TYPE STATE:
    STRUCT
        curTime: LREAL;
        dvar_M_p_vt AT %Q*: BOOL;
        dvar_M_p_vf AT %Q*: BOOL;
        dvar_M_p_vr2 AT %Q*: DINT;
        dvar_M_p_vr3 AT %Q*: DINT;
        dvar_M_p_v0 AT %Q*: DINT;
        dvar_M_p_v1 AT %Q*: DINT;
        dvar_M_p_v2 AT %Q*: DINT;
        dvar_M_p_v3 AT %Q*: DINT;
        dvar_M_p_v123 AT %Q*: DINT;
        dvar_M_p_vn1 AT %Q*: DINT;
        dvar_M_p_vn2 AT %Q*: DINT;
        dvar_M_p_v00 AT %Q*: LREAL;
        dvar_M_p_v01 AT %Q*: LREAL;
        dvar_M_p_v05 AT %Q*: LREAL;
        dvar_M_p_v10 AT %Q*: LREAL;
        dvar_M_p_v20 AT %Q*: LREAL;
        dvar_M_p_v30 AT %Q*: LREAL;
        dvar_M_p_v270 AT %Q*: LREAL;
        dvar_M_p_vn01 AT %Q*: LREAL;
        dvar_M_p_vn10 AT %Q*: LREAL;
        dvar_M_p_e AT %Q*: LREAL;
        dvar_M_p_ve1 AT %Q*: enum_E;
        dvar_M_p_ve2 AT %Q*: enum_E;
        dvar_M_p_ve3 AT %Q*: enum_E;
        dvar_M_p_ve4 AT %Q*: enum_E;
        dvar_M_p_vbir AT %Q*: TupleStruct_2;
        dvar_M_p_vb000 AT %Q*: BOOL;
        dvar_M_p_vb001 AT %Q*: BOOL;
        dvar_M_p_vb002 AT %Q*: BOOL;
        dvar_M_p_vb003 AT %Q*: BOOL;
        dvar_M_p_vb004 AT %Q*: BOOL;
        dvar_M_p_vb005 AT %Q*: BOOL;
        dvar_M_p_vb006 AT %Q*: BOOL;
        dvar_M_p_vb007 AT %Q*: BOOL;
        dvar_M_p_vb008 AT %Q*: BOOL;
        dvar_M_p_vb009 AT %Q*: BOOL;
        dvar_M_p_vb010 AT %Q*: BOOL;
        dvar_M_p_vb011 AT %Q*: BOOL;
        dvar_M_p_vb012 AT %Q*: BOOL;
        dvar_M_p_vb013 AT %Q*: BOOL;
        dvar_M_p_vb014 AT %Q*: BOOL;
        dvar_M_p_vb015 AT %Q*: BOOL;
        dvar_M_p_vb016 AT %Q*: BOOL;
        dvar_M_p_vb017 AT %Q*: BOOL;
        dvar_M_p_vb018 AT %Q*: BOOL;
        dvar_M_p_vb019 AT %Q*: BOOL;
        dvar_M_p_vb020 AT %Q*: BOOL;
        dvar_M_p_vb021 AT %Q*: BOOL;
        dvar_M_p_vb022 AT %Q*: BOOL;
        dvar_M_p_vb023 AT %Q*: BOOL;
        dvar_M_p_vb024 AT %Q*: BOOL;
        dvar_M_p_vb025 AT %Q*: BOOL;
        dvar_M_p_vb026 AT %Q*: BOOL;
        dvar_M_p_vb027 AT %Q*: BOOL;
        dvar_M_p_vb028 AT %Q*: BOOL;
        dvar_M_p_vb029 AT %Q*: BOOL;
        dvar_M_p_vb030 AT %Q*: BOOL;
        dvar_M_p_vb031 AT %Q*: BOOL;
        dvar_M_p_vb032 AT %Q*: BOOL;
        dvar_M_p_vb033 AT %Q*: BOOL;
        dvar_M_p_vb034 AT %Q*: BOOL;
        dvar_M_p_vb035 AT %Q*: BOOL;
        dvar_M_p_vb036 AT %Q*: BOOL;
        dvar_M_p_vb037 AT %Q*: BOOL;
        dvar_M_p_vb038 AT %Q*: BOOL;
        dvar_M_p_vb039 AT %Q*: BOOL;
        dvar_M_p_vb040 AT %Q*: BOOL;
        dvar_M_p_vb041 AT %Q*: BOOL;
        dvar_M_p_vb042 AT %Q*: BOOL;
        dvar_M_p_vb043 AT %Q*: BOOL;
        dvar_M_p_vb044 AT %Q*: BOOL;
        dvar_M_p_vb045 AT %Q*: BOOL;
        dvar_M_p_vb046 AT %Q*: BOOL;
        dvar_M_p_vb047 AT %Q*: BOOL;
        dvar_M_p_vb048 AT %Q*: BOOL;
        dvar_M_p_vb049 AT %Q*: BOOL;
        dvar_M_p_vb050 AT %Q*: BOOL;
        dvar_M_p_vb051 AT %Q*: BOOL;
        dvar_M_p_vb052 AT %Q*: BOOL;
        dvar_M_p_vb053 AT %Q*: BOOL;
        dvar_M_p_vb054 AT %Q*: BOOL;
        dvar_M_p_vb055 AT %Q*: BOOL;
        dvar_M_p_vb056 AT %Q*: BOOL;
        dvar_M_p_vb057 AT %Q*: BOOL;
        dvar_M_p_vb058 AT %Q*: BOOL;
        dvar_M_p_vb059 AT %Q*: BOOL;
        dvar_M_p_vb060 AT %Q*: BOOL;
        dvar_M_p_vb061 AT %Q*: BOOL;
        dvar_M_p_vb062 AT %Q*: BOOL;
        dvar_M_p_vb063 AT %Q*: BOOL;
        dvar_M_p_vb064 AT %Q*: BOOL;
        dvar_M_p_vb065 AT %Q*: BOOL;
        dvar_M_p_vb066 AT %Q*: BOOL;
        dvar_M_p_vb067 AT %Q*: BOOL;
        dvar_M_p_vb068 AT %Q*: BOOL;
        dvar_M_p_vb069 AT %Q*: BOOL;
        dvar_M_p_vb070 AT %Q*: BOOL;
        dvar_M_p_vb071 AT %Q*: BOOL;
        dvar_M_p_vb072 AT %Q*: BOOL;
        dvar_M_p_vb073 AT %Q*: BOOL;
        dvar_M_p_vb074 AT %Q*: BOOL;
        dvar_M_p_vb075 AT %Q*: BOOL;
        dvar_M_p_vb076 AT %Q*: BOOL;
        dvar_M_p_vb077 AT %Q*: BOOL;
        dvar_M_p_vb078 AT %Q*: BOOL;
        dvar_M_p_vb079 AT %Q*: BOOL;
        dvar_M_p_vb080 AT %Q*: BOOL;
        dvar_M_p_vb081 AT %Q*: BOOL;
        dvar_M_p_vb082 AT %Q*: BOOL;
        dvar_M_p_vb083 AT %Q*: BOOL;
        dvar_M_p_vb084 AT %Q*: BOOL;
        dvar_M_p_vb085 AT %Q*: BOOL;
        dvar_M_p_vb086 AT %Q*: BOOL;
        dvar_M_p_vb087 AT %Q*: BOOL;
        dvar_M_p_vb088 AT %Q*: BOOL;
        dvar_M_p_vb089 AT %Q*: BOOL;
        dvar_M_p_vb090 AT %Q*: BOOL;
        dvar_M_p_vb091 AT %Q*: BOOL;
        dvar_M_p_vb092 AT %Q*: BOOL;
        dvar_M_p_vb093 AT %Q*: BOOL;
        dvar_M_p_vb094 AT %Q*: BOOL;
        dvar_M_p_vb095 AT %Q*: BOOL;
        dvar_M_p_vb096 AT %Q*: BOOL;
        dvar_M_p_vb097 AT %Q*: BOOL;
        dvar_M_p_vb098 AT %Q*: BOOL;
        dvar_M_p_vb099 AT %Q*: BOOL;
        dvar_M_p_vi00 AT %Q*: DINT;
        dvar_M_p_vi01 AT %Q*: DINT;
        dvar_M_p_vi02 AT %Q*: DINT;
        dvar_M_p_vi03 AT %Q*: DINT;
        dvar_M_p_vi04 AT %Q*: DINT;
        dvar_M_p_vi05 AT %Q*: DINT;
        dvar_M_p_vi06 AT %Q*: DINT;
        dvar_M_p_vi07 AT %Q*: DINT;
        dvar_M_p_vi08 AT %Q*: DINT;
        dvar_M_p_vi09 AT %Q*: DINT;
        dvar_M_p_vi10 AT %Q*: DINT;
        dvar_M_p_vi11 AT %Q*: DINT;
        dvar_M_p_vi12 AT %Q*: DINT;
        dvar_M_p_vi13 AT %Q*: DINT;
        dvar_M_p_vi14 AT %Q*: DINT;
        dvar_M_p_vi15 AT %Q*: DINT;
        dvar_M_p_vi16 AT %Q*: DINT;
        dvar_M_p_vi17 AT %Q*: DINT;
        dvar_M_p_vi18 AT %Q*: DINT;
        dvar_M_p_vi19 AT %Q*: DINT;
        dvar_M_p_vi20 AT %Q*: DINT;
        dvar_M_p_vi21 AT %Q*: DINT;
        dvar_M_p_vi22 AT %Q*: DINT;
        dvar_M_p_vi23 AT %Q*: DINT;
        dvar_M_p_vi24 AT %Q*: DINT;
        dvar_M_p_vi25 AT %Q*: DINT;
        dvar_M_p_vi26 AT %Q*: DINT;
        dvar_M_p_vi27 AT %Q*: DINT;
        dvar_M_p_vi28 AT %Q*: DINT;
        dvar_M_p_vi29 AT %Q*: DINT;
        dvar_M_p_vi30 AT %Q*: DINT;
        dvar_M_p_vi31 AT %Q*: DINT;
        dvar_M_p_vi32 AT %Q*: DINT;
        dvar_M_p_vi33 AT %Q*: DINT;
        dvar_M_p_vi34 AT %Q*: DINT;
        dvar_M_p_vr00 AT %Q*: LREAL;
        dvar_M_p_vr01 AT %Q*: LREAL;
        dvar_M_p_vr02 AT %Q*: LREAL;
        dvar_M_p_vr03 AT %Q*: LREAL;
        dvar_M_p_vr04 AT %Q*: LREAL;
        dvar_M_p_vr05 AT %Q*: LREAL;
        dvar_M_p_vr06 AT %Q*: LREAL;
        dvar_M_p_vr07 AT %Q*: LREAL;
        dvar_M_p_vr08 AT %Q*: LREAL;
        dvar_M_p_vr09 AT %Q*: LREAL;
        dvar_M_p_vr10 AT %Q*: LREAL;
        dvar_M_p_vr11 AT %Q*: LREAL;
        dvar_M_p_vr12 AT %Q*: LREAL;
        dvar_M_p_vr13 AT %Q*: LREAL;
        dvar_M_p_vr14 AT %Q*: LREAL;
        dvar_M_p_vr15 AT %Q*: LREAL;
        dvar_M_p_vr16 AT %Q*: LREAL;
        dvar_M_p_vr17 AT %Q*: LREAL;
        dvar_M_p_vr18 AT %Q*: LREAL;
        dvar_M_p_vr19 AT %Q*: LREAL;
        dvar_M_p_vr20 AT %Q*: LREAL;
        dvar_M_p_vr21 AT %Q*: LREAL;
        dvar_M_p_vr22 AT %Q*: LREAL;
        dvar_M_p_vr23 AT %Q*: LREAL;
        dvar_M_p_vr24 AT %Q*: LREAL;
        dvar_M_p_vr25 AT %Q*: LREAL;
        dvar_M_p_vr26 AT %Q*: LREAL;
        dvar_M_p_vr27 AT %Q*: LREAL;
        dvar_M_p_vr28 AT %Q*: LREAL;
        dvar_M_p_vr29 AT %Q*: LREAL;
        dvar_M_p_vr30 AT %Q*: LREAL;
        dvar_M_p_vr31 AT %Q*: LREAL;
        dvar_M_p_vr32 AT %Q*: LREAL;
        dvar_M_p_vr33 AT %Q*: LREAL;
        dvar_M_p_vr34 AT %Q*: LREAL;
        dvar_M_p_vr35 AT %Q*: LREAL;
        dvar_M_p_vr36 AT %Q*: LREAL;
        dvar_M_p_vr37 AT %Q*: LREAL;
        dvar_M_p_vr38 AT %Q*: LREAL;
        dvar_M_p_vr39 AT %Q*: LREAL;
        dvar_M_p_vr40 AT %Q*: LREAL;
        dvar_M_p_vr41 AT %Q*: LREAL;
        dvar_M_p_vr42 AT %Q*: LREAL;
        dvar_M_p_vr43 AT %Q*: LREAL;
        dvar_M_p_vr44 AT %Q*: LREAL;
        dvar_M_p_vr45 AT %Q*: LREAL;
        dvar_M_p_vr46 AT %Q*: LREAL;
        dvar_M_p_vr47 AT %Q*: LREAL;
        dvar_M_p_vr48 AT %Q*: LREAL;
        dvar_M_p_vr49 AT %Q*: LREAL;
        dvar_M_p_vr50 AT %Q*: LREAL;
        dvar_M_p_vr51 AT %Q*: LREAL;
        dvar_M_p_vr52 AT %Q*: LREAL;
        dvar_M_p_vr53 AT %Q*: LREAL;
        dvar_M_p_vr54 AT %Q*: LREAL;
        dvar_M_p_vr55 AT %Q*: LREAL;
        dvar_M_p_vr56 AT %Q*: LREAL;
        dvar_M_p_vr57 AT %Q*: LREAL;
        dvar_M_p_vr58 AT %Q*: LREAL;
        dvar_M_p AT %Q*: enum_E;
    END_STRUCT
END_TYPE

(* stored: ProductVersion 3.1.0.18, Version 1.1.0.1 *)
